// TwinCAT 3 PLC project Untitled1
// ProgramVersion: 3.1.4022.4
// libraries:
//   Tc2_Standard, * (Beckhoff Automation GmbH)
//   Tc2_System, * (Beckhoff Automation GmbH)
//   Tc3_Module, * (Beckhoff Automation GmbH)
// project tree:
//   GVLs/ GVL_IO.TcGVL
//   / PlcTask.TcTTO
//   POUs/ FUN_ITR.TcPOU, MAIN.TcPOU, PWM.TcPOU
// real-time tasks:
//   TASK PlcTask: cycle T#50us, priority 20, ADS port 350
// motion (NC):
//   TASK NC-Task 1 SAF: cycle T#2ms, priority 4, ADS port 501
//   TASK NC-Task 1 SVB: cycle T#10ms, priority 8, ADS port 511
//   AXIS Axis 1 (id 1)
//     OtherSettings: AllowMotionCmdToSlave=true
//     encoder EncType=8
//       EncPara: MaxCount=#xffffffff
//     drive DrvType=9
//       DrvPara: MaxCount=#xffffffff, DriveControlDWord=#x00030100
//         Analog: VeloScale=1.02400649589962, ScaleFactorActTorque=0.1
//         TimeComp: TaskDelayCycles=1
//     controller CtrType=1
//       CtrPara: PriorControlFactor=1
//         Observer: BandWidth=20
//   AXIS Axis 2 (id 2)
//     OtherSettings: AllowMotionCmdToSlave=true
//     encoder EncType=8
//       EncPara: MaxCount=#xffffffff
//     drive DrvType=9
//       DrvPara: MaxCount=#xffffffff, DriveControlDWord=#x00030100
//         Analog: VeloScale=1.02400649589962, ScaleFactorActTorque=0.1
//         TimeComp: TaskDelayCycles=1
//     controller CtrType=1
//       CtrPara: PriorControlFactor=1
//         Observer: BandWidth=20
// I/O:
//   DEVICE Device 1 (EtherCAT), AmsNetId 169.254.89.106.2.1
//     Term 1 (EK1200) [EK1200-5000 EtherCAT Power supply (2A E-Bus)]
//       Term 2 (EL1004) [EL1004 4Ch. Dig. Input 24V, 3ms]
//       Term 3 (EL2004) [EL2004 4Ch. Dig. Output 24V, 0.5A]
//       Term 4 (EL3062) [EL3062 2Ch. Ana. Input 0-10V]
//       Term 5 (EL4002) [EL4002 2Ch. Ana. Output 0-10V, 12bit]
//       Term 6 (EK1110) [EK1110 EtherCAT extension]
//     Drive 7 (AX5203-0000-0210) [AX5203-0000-0210 EtherCAT Drive (SoE, 2 Ch.)]
// variable links:
//   NC-Task 1 SAF/Axes/Axis 1 <-> Device 1 (EtherCAT)/Drive 7 (AX5203-0000-0210)
//     Drive/Inputs/In/nDataIn1 <-> AT 1/Following distance
//     Drive/Inputs/In/nDcOutputTime <-> InfoData/DcOutputShift
//     Drive/Inputs/In/nState1 <-> AT 1/Drive status word @bit 8
//     Drive/Inputs/In/nState2 <-> AT 1/Drive status word
//     Drive/Inputs/In/nState4 @bit 1 <-> WcState/InputToggle
//     Drive/Inputs/In/nState4 <-> WcState/WcState
//     Drive/Outputs/Out/nCtrl1 <-> MDT 1/Master control word @bit 8
//     Drive/Outputs/Out/nDataOut1 <-> MDT 1/Position command value
//     Enc/Inputs/In/nDataIn1 <-> AT 1/Position feedback 1 value
//     Enc/Inputs/In/nDcInputTime <-> InfoData/DcInputShift
//     Enc/Inputs/In/nState4 @bit 1 <-> WcState/InputToggle
//     Enc/Inputs/In/nState4 <-> WcState/WcState
//   NC-Task 1 SAF/Axes/Axis 2 <-> Device 1 (EtherCAT)/Drive 7 (AX5203-0000-0210)
//     Drive/Inputs/In/nDataIn1 <-> AT 2/Following distance
//     Drive/Inputs/In/nDcOutputTime <-> InfoData/DcOutputShift
//     Drive/Inputs/In/nState1 <-> AT 2/Drive status word @bit 8
//     Drive/Inputs/In/nState2 <-> AT 2/Drive status word
//     Drive/Inputs/In/nState4 @bit 1 <-> WcState/InputToggle
//     Drive/Inputs/In/nState4 <-> WcState/WcState
//     Drive/Outputs/Out/nCtrl1 <-> MDT 2/Master control word @bit 8
//     Drive/Outputs/Out/nDataOut1 <-> MDT 2/Position command value
//     Enc/Inputs/In/nDataIn1 <-> AT 2/Position feedback 1 value
//     Enc/Inputs/In/nDcInputTime <-> InfoData/DcInputShift
//     Enc/Inputs/In/nState4 @bit 1 <-> WcState/InputToggle
//     Enc/Inputs/In/nState4 <-> WcState/WcState
//   Untitled1/Untitled1 Instance <-> Device 1 (EtherCAT)/Term 1 (EK1200)/Term 2 (EL1004)
//     PlcTask Inputs/GVL_IO.binput1 <-> Channel 1/Input
//   Untitled1/Untitled1 Instance <-> Device 1 (EtherCAT)/Term 1 (EK1200)/Term 3 (EL2004)
//     PlcTask Outputs/GVL_IO.boutput1 <-> Channel 1/Output
//   Untitled1/Untitled1 Instance <-> Device 1 (EtherCAT)/Term 1 (EK1200)/Term 4 (EL3062)
//     PlcTask Inputs/GVL_IO.ainput1 <-> AI Standard Channel 1/Value
//   Untitled1/Untitled1 Instance <-> Device 1 (EtherCAT)/Term 1 (EK1200)/Term 5 (EL4002)
//     PlcTask Outputs/GVL_IO.aoutput1 <-> AO Outputs Channel 1/Analog output

CONFIGURATION Untitled1
    RESOURCE PLC ON TwinCAT3
        TASK PlcTask(INTERVAL := T#50us, PRIORITY := 20);
        PROGRAM MAIN WITH PlcTask : MAIN;
    END_RESOURCE
END_CONFIGURATION

// ---- GVLs/GVL_IO.TcGVL
VAR_GLOBAL
	
binput1		AT%I*	:BOOL;
boutput1	AT%Q*	:BOOL;

aoutput1	AT%Q*	:INT;
ainput1		AT%I*	:INT;
END_VAR

// ---- POUs/MAIN.TcPOU
PROGRAM MAIN
VAR
	PWM1: PWM;
	tTime2: LTIME;
	a1: LREAL;
END_VAR

aoutput1:=32767;
a1:=FUN_ITR(N:=ainput1 );
tTime2:=LREAL_TO_LTIME(a1);
PWM1(bVar:=binput1 , tTime:=tTime2, Led1=>boutput1 );
pwm1.Led1;

END_PROGRAM

// ---- POUs/PWM.TcPOU
FUNCTION_BLOCK PWM
VAR_INPUT
	bVar: BOOL;
		tTime: LTIME;

END_VAR
VAR_OUTPUT
		Led1: BOOL;
END_VAR
VAR
	nState: INT;
	LTON1: LTON;
	LTON2: LTON;
	toplamT: LTIME;
	realVal1: LREAL;
	realVal2: LREAL;
	newTime: LTIME;
END_VAR

toplamT:=LTIME#200US;
realVal1:=LTIME_TO_LREAL(tTime);
realVal2:=LTIME_TO_LREAL(toplamT);

newTime:=LREAL_TO_LTIME(realVal2-realVal1);

CASE nState OF
	
0:
	IF bVar THEN
	
		nState:=10;
	
	END_IF

10:
	
	Led1:=TRUE;
	LTON1(IN:=TRUE , PT:=tTime , Q=> , ET=> );
	
	IF Lton1.Q THEN

		nState:=20;	
		LTON1(IN:=FALSE);
		
	END_IF

20:
	
	Led1:=FALSE;
	LTON2(IN:=TRUE , PT:=newTime , Q=> , ET=> );
	
	IF Lton2.Q THEN

		nState:=0;	
		LTON2(IN:=FALSE);
		
	END_IF
END_CASE

	IF NOT(bVar) THEN

		nState:=0;	
		LTON2(IN:=FALSE);
		LTON1(IN:=FALSE);

	END_IF

END_FUNCTION_BLOCK

// ---- POUs/FUN_ITR.TcPOU
FUNCTION FUN_ITR : LREAL
VAR_INPUT
	N: INT;
END_VAR
VAR
END_VAR

FUN_ITR:= (INT_TO_LREAL(N)/32767)*200000;

END_FUNCTION
